ADAPTER APickNPlace (* Adapter Interface *)
  (* Standard: 61499-1 *)
  (* Version 1.0, 2018-09-13, az *)
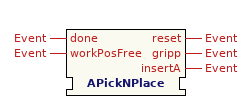
  EVENT_INPUT
    done;
    workPosFree;
  END_EVENT
  EVENT_OUTPUT
    reset;
    gripp;
    insertA;
  END_EVENT
  SERVICE SOCKET/PLUG (* Adapter Interface *)
    SEQUENCE request_confirm
      SOCKET.REQ(REQD) -> PLUG.REQ(REQD);
      PLUG.CNF(CNFD) -> SOCKET.CNF(CNFD);
    END_SEQUENCE
    SEQUENCE indication_response
      PLUG.IND(INDD) -> SOCKET.IND(INDD);
      SOCKET.RSP(RSPD) -> PLUG.RSP(RSPD);
    END_SEQUENCE
  END_SERVICE
END_ADAPTER
